// TIA Portal V19 export
TYPE "FCP_STATUS_WORD"
   STRUCT
      Reserved0 : Bool := false;
      Reserved1 : Bool := false;
      DoublePumpVgMin : Bool := false;
      PresDropCompensation : Bool := false;
      PresCmdReached : Bool := false;
      Status : Bool := false;
      Warning : Bool := false;
      Error : Bool := false;
      Reserved8 : Bool := false;
      Reserved9 : Bool := false;
      Slave : Bool := false;
      ParGroup1 : Bool := false;
      Reserved12 : Bool := false;
      Reserved13 : Bool := false;
      Reserved14 : Bool := false;
      Reserved15 : Bool := false;
   END_STRUCT;
END_TYPE
